# EPICS substitutions: db/Beckhoff_3XXX/ecmcEM3702.substitutions
file "ecmc_analogInput-chX.template"{
  pattern {CH_ID, ESLO, EOFF, EGU, PREC}
          {01, "${_ESLO=0.001}", "${_EOFF=0}", "${_EGU=bar}", "${_PREC=3}"}
          {02, "${_ESLO=0.001}", "${_EOFF=0}", "${_EGU=bar}", "${_PREC=3}"}
}

file "ecmc_status_analog-chX.template"
{
  pattern {CH_ID, KEY }
          {01,    "AI"}
          {02,    "AI"}
}
